ABB RobotStudio station: Comportamiento3.rspag

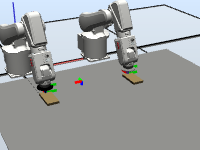
--- station ---
Station Comportamiento3 (saved by RobotStudio 6.8.8307.1040)
Controller IRB_120_dcha, task T_ROB1: task frame (RAPID world) sits at (600, 0, 0) mm, rotated rx 0 ry 0 rz -90 deg in the station
Controller IRB_120_3kg_0.58m, task T_ROB1: task frame (RAPID world) sits at (0, 0, 0) mm, rotated rx 0 ry 0 rz -90 deg in the station
Controller IRB_120_3kg_0.58m
  mechanical unit ROB_1: IRB120_izq, 6 joints, base frame (0, 0, 0) mm
Controller IRB_120_dcha
  mechanical unit ROB_1: IRB120_dcha, 6 joints, base frame (0, 0, 0) mm
Layout (positions relative to the parent item):
  - IRB120_izq [mechanism, from Robots\IRB120_3_58_G_01.rslib] at (0, 0, 0) mm, rotated rx 0 ry 0 rz -90 deg; joint values [0.0882, 1.1875, 0.0105, 0, 0.3729, 0.0882] (rad or m)
  - IRB120_dcha [mechanism, from Robots\IRB120_3_58_G_01.rslib] at (600, 0, 0) mm, rotated rx 0 ry 0 rz -90 deg; joint values [0.0882, 1.1864, 0.0111, 0, 0.3733, 0.0882] (rad or m)
  - suelo [part] at (-316.08, -1334.54, 0) mm
  - Herramienta_izda [mechanism] at (37.5, -423.96, 63.24) mm, rotated rx -180 ry 0 rz 90 deg
      TCP Herramienta_izda at (0, 0, 43.24) mm
      links: Herramienta_izda
  - Herramienta_dcha [mechanism] at (637.49, -423.96, 63.58) mm, rotated rx 180 ry 0 rz 90 deg
      TCP Herramientaa_dcha at (0, 0.01, 43.58) mm
      links: Herramienta_dcha
  - Attacher [smart component, from Components\Attacher.rslib]
      properties: Parent=IRB120_dcha; Flange=0; Child=Pieza1_dcha; Mount=false; Offset=[0 0 0]; Orientation=[0 0 0]
  - Detacher [smart component, from Components\Detacher.rslib]
      properties: Child=Pieza1_dcha; KeepPosition=true
  - LogicGate [smart component, from Components\LogicGate.rslib]
      properties: Operator=NOT; Delay=0
  - Queue [smart component, from Components\Queue.rslib]
      properties: Back=Pieza6_dcha; Front=Pieza1_dcha; Queue={9e2edeae-7e64-4a9f-bdc8-63d7fd2045a9};{d88fa062-0d92-45d6-b1ae-3425f0cffda4};{c1e01d27-fe17-4096-be87-61ebd46bfd3f};{a1d0ce36-37ec-423f-9baf-c3239c14e9f5};{bdc3ae6c-ab91-499e-a480-f0fe7d4a7228};{bc8c10a8-22dc-443d-877a-0e593dbc9cae}; NumberOfObjects=6
  - Queue_2 [smart component, from Components\Queue.rslib]
      properties: Back=Pieza6_izda; Front=Pieza1_izda; Queue={cdf0cd76-90c6-44b7-b2f9-a42f506c648d};{2fc02efc-64a9-40b3-a3fe-42393960ad30};{197146fa-7a9f-4a58-b703-2abc433c9011};{d93c40ad-8283-40ad-a29a-25ba7441558d};{0ca880e8-362b-4b33-950d-3b7a9688107a};{e9f17f10-0b3b-4bc2-a77a-605db1a7ee61}; NumberOfObjects=6
  - Attacher_2 [smart component, from Components\Attacher.rslib]
      properties: Parent=IRB120_izq; Flange=0; Child=Pieza1_izda; Mount=false; Offset=[0 0 0]; Orientation=[0 0 0]
  - LogicGate_2 [smart component, from Components\LogicGate.rslib]
      properties: Operator=NOT; Delay=0
  - Logger [smart component, from Components\Logger.rslib]
      properties: Format=wwwww; Message=wwwww; Severity=0
  - Logger_2 [smart component, from Components\Logger.rslib]
      properties: Format=nottttt; Message=nottttt; Severity=0
  - Logger_4 [smart component, from Components\Logger.rslib]
      properties: Format=d11; Message=d11; Severity=0
  - Detacher_5 [smart component, from Components\Detacher.rslib]
      properties: Child=Pieza1_izda; KeepPosition=true
  - Pieza2_dcha [part] at (600, -461.46, 5) mm
  - Pieza1_dcha [part] at (600, -436.46, 5) mm
  - Pieza3_dcha [part] at (600, -486.46, 5) mm
  - Pieza4_dcha [part] at (600, -511.46, 5) mm
  - Pieza5_dcha [part] at (600, -536.46, 5) mm
  - Pieza2_izda [part] at (0, -461.46, 5) mm
  - Pieza6_dcha [part] at (600, -561.46, 5) mm
  - Pieza1_izda [part] at (0, -436.46, 5) mm
  - Pieza3_izda [part] at (0, -486.46, 5) mm
  - Pieza4_izda [part] at (0, -511.46, 5) mm
  - Pieza5_izda [part] at (0, -536.46, 5) mm
  - Pieza6_izda [part] at (0, -561.46, 5) mm
Attachment: Herramienta_izda is attached to IRB120_izq / Link6
Attachment: Herramienta_dcha is attached to IRB120_dcha / Link6
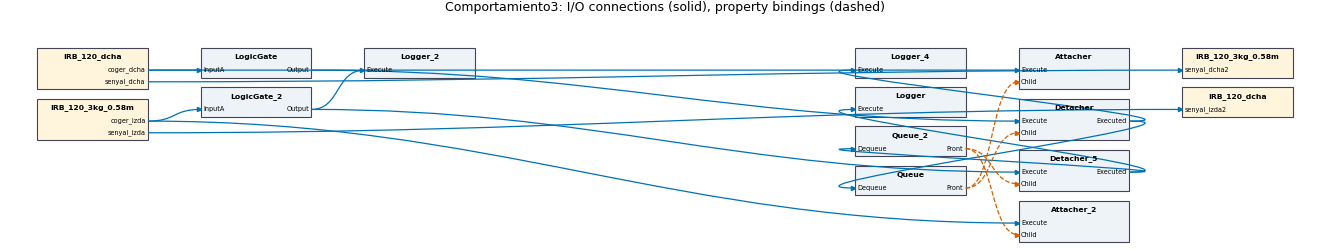
Station logic (signal -> signal, property => property):
  IRB_120_dcha.coger_dcha -> Attacher.Execute
  IRB_120_dcha.coger_dcha -> LogicGate.InputA
  LogicGate.Output -> Detacher.Execute
  IRB_120_3kg_0.58m.coger_izda -> LogicGate_2.InputA
  IRB_120_3kg_0.58m.coger_izda -> Attacher_2.Execute
  IRB_120_dcha.senyal_dcha -> IRB_120_3kg_0.58m.senyal_dcha2
  IRB_120_3kg_0.58m.senyal_izda -> IRB_120_dcha.senyal_izda2
  LogicGate_2.Output -> Logger_2.Execute
  Detacher.Executed -> Logger_4.Execute
  LogicGate_2.Output -> Detacher_5.Execute
  Detacher_5.Executed -> Logger.Execute
  Detacher_5.Executed -> Queue_2.Dequeue
  Detacher.Executed -> Queue.Dequeue
  Queue.Front => Attacher.Child
  Queue.Front => Detacher.Child
  Queue_2.Front => Attacher_2.Child
  Queue_2.Front => Detacher_5.Child

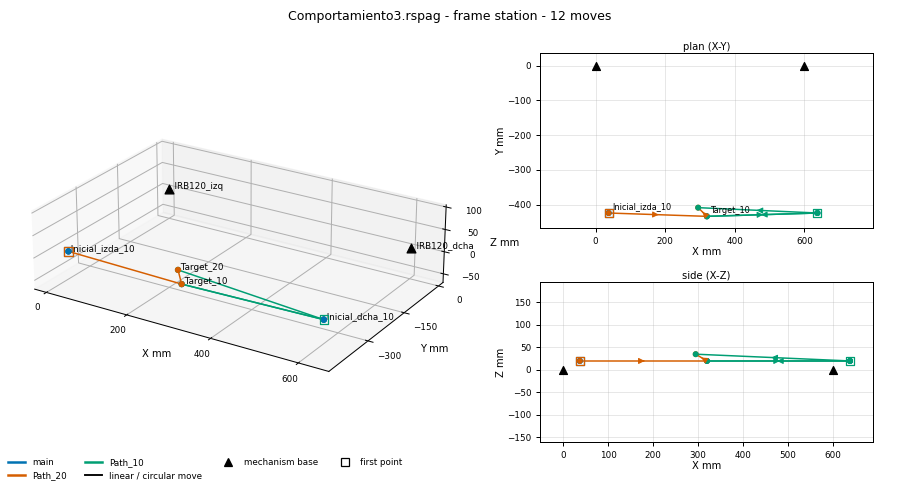
[picture p0: tool path of Comportamiento3.rspag in frame station, 12 of 59 moves have a stored position in this frame; points joined in program order, loops and branches not executed]
--- Backups/IRB_120_3kg_0.58m/RAPID/TASK1/PROGMOD/CalibData.mod ---
MODULE CalibData
	PERS tooldata MyTool:=[TRUE,[[31.7926,0,229.639],[0.945519,0,0.325568,0]],[1,[0,0,1],[1,0,0,0],0,0,0]];
	PERS tooldata Herramienta_izda:=[TRUE,[[0,0,43.241],[1,0,0,0]],[1,[0,0,1],[1,0,0,0],0,0,0]];
ENDMODULE

--- Backups/IRB_120_3kg_0.58m/RAPID/TASK1/PROGMOD/Module1.mod ---
MODULE Module1
    CONST robtarget Inicio_izda:=[[433.57,15.136,17.301],[0,0,1,0],[0,0,-1,0],[9E+09,9E+09,9E+09,9E+09,9E+09,9E+09]];
    CONST robtarget Target_10:=[[433.57,319.8,20],[0,0,1,0],[0,0,0,0],[9E+09,9E+09,9E+09,9E+09,9E+09,9E+09]];

VAR num x := 0;
VAR num y := 0;
VAR num z := 0;
	CONST robtarget Inicial_izda_10:=[[423.958,37.5,20],[0,0,1,0],[0,0,0,0],[9E+09,9E+09,9E+09,9E+09,9E+09,9E+09]];
    CONST robtarget Target_20:=[[408.57,294.8,35],[0,-0.707106781,0.707106781,0],[0,0,0,0],[9E+09,9E+09,9E+09,9E+09,9E+09,9E+09]];


    !***********************************************************
    !
    ! Módulo:  Module1
    !
    ! Descripción:
    !   <Introduzca la descripción aquí>
    !
    ! Autor: Nicolás
    !
    ! Versión: 1.0
    !
    !***********************************************************


    !***********************************************************
    !
    ! Procedimiento Main
    !
    !   Este es el punto de entrada de su programa
    !
    !***********************************************************
    PROC main()

        ! Movimiento del otro robot
        MoveL offs(Inicial_izda_10,x,y,20),v200,fine,Herramienta_izda\WObj:=wobj0;
        reset senyal_izda;
        WaitTime(1);
        WaitDI senyal_dcha2,1;

        ! PRIMER BLOQUE

        MoveL offs(Inicial_izda_10,x,y,20),v200,fine,Herramienta_izda\WObj:=wobj0;
        waittime(1);
        MoveL Inicial_izda_10,v200,fine,Herramienta_izda\WObj:=wobj0;
        setdo coger_izda,1;

        x := x - 25;
        MoveL offs(Target_10,x,y,20),v100,fine,Herramienta_izda\WObj:=wobj0;
        MoveL offs(Target_10,x,y,z),v100,fine,Herramienta_izda\WObj:=wobj0;
        setdo coger_izda,0;
        reset coger_izda;
        x := 0;
        x := x + 25;
        MoveL offs(Inicial_izda_10,x,y,20),v200,fine,Herramienta_izda\WObj:=wobj0;

        ! Movimiento del otro robot
        setdo senyal_izda,1;
        WaitTime(1);
        WaitDI senyal_dcha2,1;
        setdo senyal_izda, 0;

        ! SEGUNDO BLOQUE
        MoveL offs(Inicial_izda_10,x,y,z),v200,fine,Herramienta_izda\WObj:=wobj0;
        setdo coger_izda, 1;
        x := 0;
        MoveL offs(Target_20,x,y,20),v200,fine,Herramienta_izda\WObj:=wobj0;
        MoveL offs(Target_20,x,y,z),v200,fine,Herramienta_izda\WObj:=wobj0;
        setdo coger_izda,0;

        x := x + 50;
        MoveL offs(Inicial_izda_10,x,y,20),v200,fine,Herramienta_izda\WObj:=wobj0;

        ! Movimiento del otro robot
        setdo senyal_izda,1;
        WaitTime(1);
        WaitDI senyal_dcha2,1;
        setdo senyal_izda, 0;

        ! TERCER BLOQUE
        MoveL offs(Inicial_izda_10,x,y,z),v200,fine,Herramienta_izda\WObj:=wobj0;
        setdo coger_izda, 1;
        x := 0;
        y := 50;
        MoveL offs(Target_20,x,y,20),v200,fine,Herramienta_izda\WObj:=wobj0;
        MoveL offs(Target_20,x,y,z),v200,fine,Herramienta_izda\WObj:=wobj0;
        setdo coger_izda,0;
        y := 0;
        x := 75;
        MoveL offs(Inicial_izda_10,x,y,20),v200,fine,Herramienta_izda\WObj:=wobj0;

        ! Movimiento del otro robot
        setdo senyal_izda,1;
        WaitTime(1);
        WaitDI senyal_dcha2,1;
        setdo senyal_izda, 0;

        ! CUARTO BLOQUE
        MoveL offs(Inicial_izda_10,x,y,z),v200,fine,Herramienta_izda\WObj:=wobj0;
        setdo coger_izda, 1;
        x := 0;
        x := x - 25;
        MoveL offs(Target_10,x,y,50),v200,fine,Herramienta_izda\WObj:=wobj0;
        MoveL offs(Target_10,x,y,30),v200,fine,Herramienta_izda\WObj:=wobj0;
        setdo coger_izda,0;

        x := 100;
        MoveL offs(Inicial_izda_10,x,y,20),v200,fine,Herramienta_izda\WObj:=wobj0;

        ! Movimiento del otro robot
        setdo senyal_izda,1;
        WaitTime(1);
        WaitDI senyal_dcha2,1;
        setdo senyal_izda, 0;

        ! QUINTO BLOQUE
        MoveL offs(Inicial_izda_10,x,y,z),v200,fine,Herramienta_izda\WObj:=wobj0;
        setdo coger_izda, 1;
        x := 0;
        MoveL offs(Target_20,x,y,50),v200,fine,Herramienta_izda\WObj:=wobj0;
        MoveL offs(Target_20,x,y,30),v200,fine,Herramienta_izda\WObj:=wobj0;
        setdo coger_izda,0;

        x := 125;
        MoveL offs(Inicial_izda_10,x,y,20),v200,fine,Herramienta_izda\WObj:=wobj0;

        ! Movimiento del otro robot
        setdo senyal_izda,1;
        WaitTime(1);
        WaitDI senyal_dcha2,1;
        setdo senyal_izda, 0;

        ! SEXTO BLOQUE
        MoveL offs(Inicial_izda_10,x,y,z),v200,fine,Herramienta_izda\WObj:=wobj0;
        setdo coger_izda, 1;
        y := 50;
        x := 0;
        MoveL offs(Target_20,x,y,50),v200,fine,Herramienta_izda\WObj:=wobj0;
        MoveL offs(Target_20,x,y,30),v200,fine,Herramienta_izda\WObj:=wobj0;
        setdo coger_izda,0;

        MoveL Inicial_izda_10,v200,fine,Herramienta_izda\WObj:=wobj0;


    ENDPROC
    PROC Path_20()
        MoveL Inicial_izda_10,v200,z100,Herramienta_izda\WObj:=wobj0;
        MoveL Target_10,v200,z100,Herramienta_izda\WObj:=wobj0;
        MoveL Target_20,v200,fine,Herramienta_izda\WObj:=wobj0;
    ENDPROC
!    PROC Path_20()
!        MoveL Inicial_izda_10,v200,z100,Herramienta_izda\WObj:=wobj0;
!		MoveL Target_10,v200,z100,Herramienta_izda\WObj:=wobj0;
!        MoveL Target_20,v200,fine,Herramienta_izda\WObj:=wobj0;
!    ENDPROC
!    PROC Path_30()
!        MoveL Target_10,v1000,z100,Herramienta_izda\WObj:=wobj0;
!    ENDPROC
ENDMODULE

--- Backups/IRB_120_dcha/RAPID/TASK1/PROGMOD/CalibData.mod ---
MODULE CalibData
	PERS tooldata MyTool:=[TRUE,[[31.7926,0,229.639],[0.945519,0,0.325568,0]],[1,[0,0,1],[1,0,0,0],0,0,0]];
	PERS tooldata Herramientaa_dcha:=[TRUE,[[0,0.014,43.581],[1,0,0,0]],[1,[0,0,1],[1,0,0,0],0,0,0]];
ENDMODULE

--- Backups/IRB_120_dcha/RAPID/TASK1/PROGMOD/Module1.mod ---
MODULE Module1
	CONST robtarget Inicio_dcha:=[[432.307,18.416,18.404],[0,0,1,0],[0,-1,0,0],[9E+09,9E+09,9E+09,9E+09,9E+09,9E+09]];

VAR num x := 0;
VAR num y := 0;
VAR num z := 0;
	CONST robtarget Target_10:=[[433.57,-280.2,20],[0,0,1,0],[0,0,0,0],[9E+09,9E+09,9E+09,9E+09,9E+09,9E+09]];
    CONST robtarget Inicial_dcha_10:=[[423.958,37.5,20],[0,0,1,0],[0,0,0,0],[9E+09,9E+09,9E+09,9E+09,9E+09,9E+09]];
    CONST robtarget Target_20:=[[408.57,-305.2,35],[0,-0.707106781,0.707106781,0],[-1,0,-2,0],[9E+09,9E+09,9E+09,9E+09,9E+09,9E+09]];

    !***********************************************************
    !
    ! Módulo:  Module1
    !
    ! Descripción:
    !   <Introduzca la descripción aquí>
    !
    ! Autor: Nicolás
    !
    ! Versión: 1.0
    !
    !***********************************************************


    !***********************************************************
    !
    ! Procedimiento Main
    !
    !   Este es el punto de entrada de su programa
    !
    !***********************************************************
    PROC main()

        MoveL offs(Inicial_dcha_10,x,y,20),v200,fine,Herramientaa_dcha\WObj:=wobj0;
        Reset senyal_dcha;

        ! PRIMER BLOQUE
        MoveL offs(Inicial_dcha_10,x,y,20),v200,fine,Herramientaa_dcha\WObj:=wobj0;
        MoveL Inicial_dcha_10,v200,fine,Herramientaa_dcha\WObj:=wobj0;
        setDo coger_dcha, 1;
        MoveL offs(Target_10,y,z,20),v100,fine,Herramientaa_dcha\WObj:=wobj0;
        MoveL Target_10,v100,fine,Herramientaa_dcha\WObj:=wobj0;
        setdo coger_dcha, 0;

        x := 0;
        x := x + 25;
        MoveL offs(Inicial_dcha_10,x,y,20),v200,fine,Herramientaa_dcha\WObj:=wobj0;
        ! -----------
        ! Movimiento del otro robot
        setdo senyal_dcha,1;
        WaitTime(1);
        WaitDI senyal_izda2,1;
        setdo senyal_dcha, 0;

        ! SEGUNDO BLOQUE
        MoveL offs(Inicial_dcha_10,x,y,z),v200,fine,Herramientaa_dcha\WObj:=wobj0;
        setDo coger_dcha, 1;
        x := 0;
        x := x - 50;
        MoveL offs(Target_10,x,y,20),v100,fine,Herramientaa_dcha\WObj:=wobj0;
        MoveL offs(Target_10,x,y,z),v100,fine,Herramientaa_dcha\WObj:=wobj0;
        setdo coger_dcha, 0;

        x := 0;
        x := x + 50;
        MoveL offs(Inicial_dcha_10,x,y,20),v200,fine,Herramientaa_dcha\WObj:=wobj0;


        ! Movimiento del otro robot
        setdo senyal_dcha,1;
        WaitTime(1);
        WaitDI senyal_izda2,1;
        Reset senyal_dcha;

        ! TERCER BLOQUE
        MoveL offs(Inicial_dcha_10,x,y,z),v200,fine,Herramientaa_dcha\WObj:=wobj0;
        setdo coger_dcha, 1;
        x := 0;
        y := y + 25;
        MoveL offs(Target_20,x,y,20),v200,fine,Herramientaa_dcha\WObj:=wobj0;
        MoveL offs(Target_20,x,y,z),v200,fine,Herramientaa_dcha\WObj:=wobj0;
        setdo coger_dcha, 0;
        y := 0;
        x := 0;
        x := x + 75;
        MoveL offs(Inicial_dcha_10,x,y,20),v200,fine,Herramientaa_dcha\WObj:=wobj0;

        ! Movimiento del otro robot
        setdo senyal_dcha,1;
        WaitTime(1);
        WaitDI senyal_izda2,1;
        Reset senyal_dcha;

        ! CUARTO BLOQUE
        MoveL offs(Inicial_dcha_10,x,y,z),v200,fine,Herramientaa_dcha\WObj:=wobj0;
        setdo coger_dcha,1;
        x := 0;
        MoveL offs(Target_10,x,y,50),v100,fine,Herramientaa_dcha\WObj:=wobj0;
        MoveL offs(Target_10,x,y,30),v100,fine,Herramientaa_dcha\WObj:=wobj0;
        setdo coger_dcha, 0;


        x := x + 100;
        MoveL offs(Inicial_dcha_10,x,y,20),v200,fine,Herramientaa_dcha\WObj:=wobj0;

        ! Movimiento del otro robot
        setdo senyal_dcha,1;
        WaitTime(1);
        WaitDI senyal_izda2,1;
        Reset senyal_dcha;

        ! QUINTO BLOQUE
        MoveL offs(Inicial_dcha_10,x,y,z),v200,fine,Herramientaa_dcha\WObj:=wobj0;
        setdo coger_dcha, 1;
        x := -50;
        MoveL offs(Target_10,x,y,50),v100,fine,Herramientaa_dcha\WObj:=wobj0;
        MoveL offs(Target_10,x,y,30),v100,fine,Herramientaa_dcha\WObj:=wobj0;
        setdo coger_dcha, 0;

        x := 0;
        x := x + 125;
        MoveL offs(Inicial_dcha_10,x,y,20),v200,fine,Herramientaa_dcha\WObj:=wobj0;

        ! Movimiento del otro robot
        setdo senyal_dcha,1;
        WaitTime(1);
        WaitDI senyal_izda2,1;
        Reset senyal_dcha;

        ! SEXTO BLOQUE
        MoveL offs(Inicial_dcha_10,x,y,z),v200,fine,Herramientaa_dcha\WObj:=wobj0;
        setdo coger_dcha, 1;
        x := 0;
        y := +25;
        MoveL offs(Target_20,x,y,50),v200,fine,Herramientaa_dcha\WObj:=wobj0;
        MoveL offs(Target_20,x,y,30),v200,fine,Herramientaa_dcha\WObj:=wobj0;
        setdo coger_dcha, 0;

        ! FIN
        MoveL Inicial_dcha_10,v200,fine,Herramientaa_dcha\WObj:=wobj0;

        ! Movimiento del otro robot
        setdo senyal_dcha,1;
        WaitTime(1);
        WaitDI senyal_izda2,1;
        Reset senyal_dcha;



    ENDPROC
	PROC Path_10()
        MoveL Inicial_dcha_10,v200,fine,Herramientaa_dcha\WObj:=wobj0;
        MoveL Target_10,v200,fine,Herramientaa_dcha\WObj:=wobj0;
        MoveL Inicial_dcha_10,v1000,z100,Herramientaa_dcha\WObj:=wobj0;
        MoveL Target_20,v200,fine,Herramientaa_dcha\WObj:=wobj0;


    ENDPROC
ENDMODULE

--- Backups/IRB_120_3kg_0.58m/SYSPAR/EIO.cfg ---
EIO:CFG_1.0:6:1::
#
EIO_SIGNAL:

      -Name "coger_izda" -SignalType "DO"

      -Name "senyal_dcha2" -SignalType "DI"

      -Name "senyal_izda" -SignalType "DO"

--- Backups/IRB_120_dcha/SYSPAR/EIO.cfg ---
EIO:CFG_1.0:6:1::
#
EIO_SIGNAL:

      -Name "coger_dcha" -SignalType "DO"

      -Name "senyal_dcha" -SignalType "DO"

      -Name "senyal_izda2" -SignalType "DI"
